Staubli VAL3: SetProerty.pgx

public program SetProerty(string x_sTitle, num x_nTopX, num x_nTopY, num x_nBottomX, num x_nBottomY, string& x_sListItem[], string& x_sItem)
  local num l_nKey
  local num l_nItem
  local string l_sTemp
begin
  call setSizeList(x_nTopX,x_nTopY,x_nBottomX,x_nBottomY)
  call listcreate(x_sTitle)
  call listadd(x_sListItem)
  call listupdate(0)
  call clear(0,13)
  call typeMenu(1,"OK")
  l_sTemp=x_sItem
  do
    l_nKey=getKey()
    call listevent(l_nKey,l_nItem,x_sItem)
    delay(0)
  until l_nKey==271 or l_nKey==255 or l_nKey==270
  if l_nKey==255
    x_sItem=l_sTemp
  endIf
  wait(getKey()==-1)
end
